DATA_BLOCK "ST10_Flow14_B2Press_iDB"
{ S7_Optimized_Access := 'TRUE' }
VERSION : 0.1
NON_RETAIN
// ATTRIBUTES
// AUTO_NUMBER = False
// BLOCK_NUMBER = 1084
// END_ATTRIBUTES
"ST10_Flow14_B2Press"

BEGIN

END_DATA_BLOCK

